Staubli VAL3: CloseFile.pgx

public program CloseFile()
begin
  $fileClose(nFileHandle)
  $fileClose(0)
  $fileClose(1)
  $fileClose(2)
  $fileClose(3)
  $fileClose(4)
  $fileClose(5)
  $fileClose(6)
  $fileClose(7)
  $fileClose(8)
  $fileClose(9)
end
